// TIA Portal V18 export
// export: Created 2025-12-01T12:38:33.2765069Z, ExportSetting None, DisplayName Totally Integrated Automation Portal, DisplayVersion V18 Update 5, DisplayName TIA Portal Openness, DisplayVersion V18 Update 5, DisplayName TIA Portal Teamcenter Gateway, DisplayVersion V18, DisplayName TIA Portal Version Control Interface, DisplayVersion V18, DisplayName STEP 7 Professional, DisplayVersion V18 Update 5, DisplayName STEP 7 Safety, DisplayVersion V18, DisplayName WinCC Professional, DisplayVersion V18 Update 5
FUNCTION "ST10Cyl_interface1-10" : Void   // FC1020, LAD
{ S7_Optimized_Access := 'FALSE' }
// stored: AutoNumber false, SetENOAutomatically false
   VAR_INPUT
      AlwaysON : Bool;
      E_stop : Bool;
   END_VAR
   VAR_TEMP
      tTest : Bool;
      i : Int;
   END_VAR
BEGIN

REGION Network 1 (SCL): Cylinder 1-10 IO Interface (SCL)
   IF "Station_Sys".Manual.Mode THEN

       FOR #i := 1 TO 100 BY 1

       DO
           "ST10Cylinder".Cy[#i].In.ManualOutputType := TRUE;

       END_FOR;

   END_IF;

   //Cylinder1 IO  A-Loading-01HorizontalCylinder
   //Input
   "ST10Cylinder".Cy[1].In.WorkPositionSensor := "iA-Loading-01HorizontalCylinderInWP";
   "ST10Cylinder".Cy[1].In.HomePositionSensor := "iA-Loading-01HorizontalCylinderInHP";
   //Output
   "oA-Loading-01HorizontalCylinderToWP" := "ST10Cylinder".Cy[1].Out.GoWorkPosition;
   "oA-Loading-01HorizontalCylinderToHP" := "ST10Cylinder".Cy[1].Out.GoHomePosition;

   //Cylinder2 IO  A-Loading-01UpDownTakeCylinder
   //Input
   "ST10Cylinder".Cy[2].In.WorkPositionSensor := "iA-Loading-01UpDownTakeCylinderInWP";
   "ST10Cylinder".Cy[2].In.HomePositionSensor := "iA-Loading-01UpDownTakeCylinderInHP";
   //Output
   "oA-Loading-01UpDownTakeCylinderToWP" := "ST10Cylinder".Cy[2].Out.GoWorkPosition;
   "oA-Loading-01UpDownTakeCylinderToHP" := "ST10Cylinder".Cy[2].Out.GoHomePosition;

   //Cylinder3 IO  A-Loading-02HorizontalCylinder
   //Input
   "ST10Cylinder".Cy[3].In.WorkPositionSensor := "iA-Loading-02HorizontalCylinderInWP"  ;
   "ST10Cylinder".Cy[3].In.HomePositionSensor := "iA-Loading-02HorizontalCylinderInHP"  ;
   //Output
   "oA-Loading-02HorizontalCylinderToWP" := "ST10Cylinder".Cy[3].Out.GoWorkPosition;
   "oA-Loading-02HorizontalCylinderToHP" := "ST10Cylinder".Cy[3].Out.GoHomePosition;

   //Cylinder4 IO     A-Loading-02UpDownTakeCylinder
   //Input
   "ST10Cylinder".Cy[4].In.WorkPositionSensor := "iA-Loading-02UpDownTakeCylinderInWP";
   "ST10Cylinder".Cy[4].In.HomePositionSensor := "iA-Loading-02UpDownTakeCylinderInHP";
   //Output
   "oA-Loading-02UpDownTakeCylinderToWP" := "ST10Cylinder".Cy[4].Out.GoWorkPosition;
   "oA-Loading-02UpDownTakeCylinderToHP" := "ST10Cylinder".Cy[4].Out.GoHomePosition;

   //Cylinder5 IO  B-PressFitting-01GripperCylinder
   //Input
   "ST10Cylinder".Cy[5].In.WorkPositionSensor := "iB-PressFitting-01GripperCylinderInWP";
   "ST10Cylinder".Cy[5].In.HomePositionSensor := "iB-PressFitting-01GripperCylinderInHP";
   //Output
   "oB-PressFitting-01GripperCylinderToWP" := "ST10Cylinder".Cy[5].Out.GoWorkPosition;
   "oB-PressFitting-01GripperCylinderToHP" := "ST10Cylinder".Cy[5].Out.GoHomePosition;

   //Cylinder6 IO  B-PressFitting-01Cylinder
   //Input
   "ST10Cylinder".Cy[6].In.WorkPositionSensor := "iB-PressFitting-01CylinderInWP" ;
   "ST10Cylinder".Cy[6].In.HomePositionSensor := "iB-PressFitting-01CylinderInHP" ;
   //Output
   "oB-PressFitting-01CylinderToWP" := "ST10Cylinder".Cy[6].Out.GoWorkPosition;
   "oB-PressFitting-01CylinderToHP" := "ST10Cylinder".Cy[6].Out.GoHomePosition;

   //Cylinder7 IO  B-PressFitting-02GripperCylinder
   //Input
   "ST10Cylinder".Cy[7].In.WorkPositionSensor := "iB-PressFitting-02GripperCylinderInWP";
   "ST10Cylinder".Cy[7].In.HomePositionSensor := "iB-PressFitting-02GripperCylinderInHP";
   //Output
   "oB-PressFitting-02GripperCylinderToWP" := "ST10Cylinder".Cy[7].Out.GoWorkPosition;
   "oB-PressFitting-02GripperCylinderToHP" := "ST10Cylinder".Cy[7].Out.GoHomePosition;

   //Cylinder8 IO  B-PressFitting-02Cylinder
   //Input
   "ST10Cylinder".Cy[8].In.WorkPositionSensor := "iB-PressFitting-02CylinderInWP";
   "ST10Cylinder".Cy[8].In.HomePositionSensor := "iB-PressFitting-02CylinderInHP";
   //Output
   "oB-PressFitting-02CylinderToWP" := "ST10Cylinder".Cy[8].Out.GoWorkPosition;
   "oB-PressFitting-02CylinderToHP" := "ST10Cylinder".Cy[8].Out.GoHomePosition;

   //Cylinder9 IO  C-LocationCylinder
   //Input
   "ST10Cylinder".Cy[9].In.WorkPositionSensor := "iC-LocationCylinderInWP";
   "ST10Cylinder".Cy[9].In.HomePositionSensor := "iC-LocationCylinderInHP";
   //Output
   "oC-LocationCylinderToWP" := "ST10Cylinder".Cy[9].Out.GoWorkPosition;
   "oC-LocationCylinderToHP" := "ST10Cylinder".Cy[9].Out.GoHomePosition;


   //Cylinder10 IO  Spare
   //Input
   "ST10Cylinder".Cy[10].In.WorkPositionSensor := "ST10Cylinder".Cy[10].Out.GoWorkPosition ;
   "ST10Cylinder".Cy[10].In.HomePositionSensor := "ST10Cylinder".Cy[10].Out.GoHomePosition ;
   //Output
   "ST10Cylinder".Cy[10].Out.GoWorkPosition := "ST10Cylinder".Cy[10].Out.GoWorkPosition;
   "ST10Cylinder".Cy[10].Out.GoHomePosition := "ST10Cylinder".Cy[10].Out.GoHomePosition;
END_REGION

REGION Network 2: CY1 interface A-Loading-01HorizontalCylinder
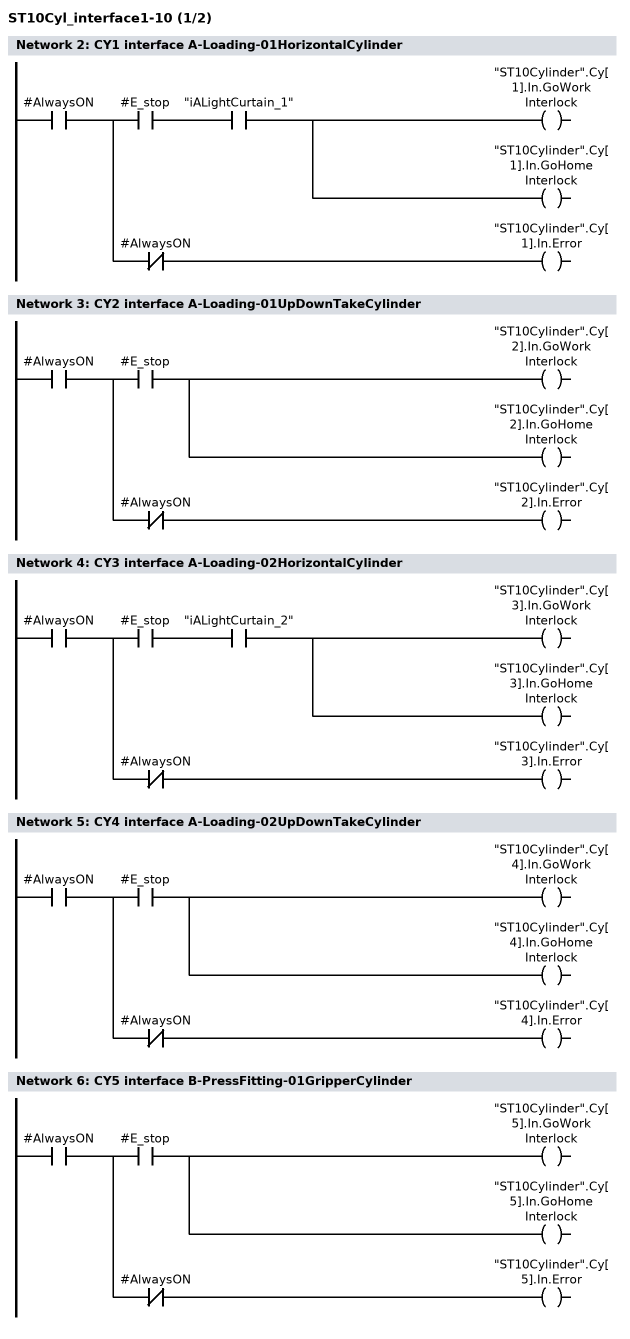
   RUNG wire#powerrail
      Contact( #AlwaysON )
      wire#w1
      Contact( #E_stop )
      Contact( "iALightCurtain_1" )
      wire#w2
      Coil( "ST10Cylinder".Cy[1].In.GoWorkInterlock )
   END_RUNG
   RUNG wire#w2
      Coil( "ST10Cylinder".Cy[1].In.GoHomeInterlock )
   END_RUNG
   RUNG wire#w1
      I_Contact( #AlwaysON )
      Coil( "ST10Cylinder".Cy[1].In.Error )
   END_RUNG
   // the same network as SCL:
   "ST10Cylinder".Cy[1].In.GoWorkInterlock := #AlwaysON AND #E_stop AND "iALightCurtain_1";
   "ST10Cylinder".Cy[1].In.GoHomeInterlock := #AlwaysON AND #E_stop AND "iALightCurtain_1";
   "ST10Cylinder".Cy[1].In.Error := #AlwaysON AND NOT #AlwaysON;
END_REGION

REGION Network 3: CY2 interface A-Loading-01UpDownTakeCylinder
   RUNG wire#powerrail
      Contact( #AlwaysON )
      wire#w1
      Contact( #E_stop )
      wire#w2
      Coil( "ST10Cylinder".Cy[2].In.GoWorkInterlock )
   END_RUNG
   RUNG wire#w2
      Coil( "ST10Cylinder".Cy[2].In.GoHomeInterlock )
   END_RUNG
   RUNG wire#w1
      I_Contact( #AlwaysON )
      Coil( "ST10Cylinder".Cy[2].In.Error )
   END_RUNG
   // the same network as SCL:
   "ST10Cylinder".Cy[2].In.GoWorkInterlock := #AlwaysON AND #E_stop;
   "ST10Cylinder".Cy[2].In.GoHomeInterlock := #AlwaysON AND #E_stop;
   "ST10Cylinder".Cy[2].In.Error := #AlwaysON AND NOT #AlwaysON;
END_REGION

REGION Network 4: CY3 interface A-Loading-02HorizontalCylinder
   RUNG wire#powerrail
      Contact( #AlwaysON )
      wire#w1
      Contact( #E_stop )
      Contact( "iALightCurtain_2" )
      wire#w2
      Coil( "ST10Cylinder".Cy[3].In.GoWorkInterlock )
   END_RUNG
   RUNG wire#w2
      Coil( "ST10Cylinder".Cy[3].In.GoHomeInterlock )
   END_RUNG
   RUNG wire#w1
      I_Contact( #AlwaysON )
      Coil( "ST10Cylinder".Cy[3].In.Error )
   END_RUNG
   // the same network as SCL:
   "ST10Cylinder".Cy[3].In.GoWorkInterlock := #AlwaysON AND #E_stop AND "iALightCurtain_2";
   "ST10Cylinder".Cy[3].In.GoHomeInterlock := #AlwaysON AND #E_stop AND "iALightCurtain_2";
   "ST10Cylinder".Cy[3].In.Error := #AlwaysON AND NOT #AlwaysON;
END_REGION

REGION Network 5: CY4 interface A-Loading-02UpDownTakeCylinder
   RUNG wire#powerrail
      Contact( #AlwaysON )
      wire#w1
      Contact( #E_stop )
      wire#w2
      Coil( "ST10Cylinder".Cy[4].In.GoWorkInterlock )
   END_RUNG
   RUNG wire#w2
      Coil( "ST10Cylinder".Cy[4].In.GoHomeInterlock )
   END_RUNG
   RUNG wire#w1
      I_Contact( #AlwaysON )
      Coil( "ST10Cylinder".Cy[4].In.Error )
   END_RUNG
   // the same network as SCL:
   "ST10Cylinder".Cy[4].In.GoWorkInterlock := #AlwaysON AND #E_stop;
   "ST10Cylinder".Cy[4].In.GoHomeInterlock := #AlwaysON AND #E_stop;
   "ST10Cylinder".Cy[4].In.Error := #AlwaysON AND NOT #AlwaysON;
END_REGION

REGION Network 6: CY5 interface B-PressFitting-01GripperCylinder
   RUNG wire#powerrail
      Contact( #AlwaysON )
      wire#w1
      Contact( #E_stop )
      wire#w2
      Coil( "ST10Cylinder".Cy[5].In.GoWorkInterlock )
   END_RUNG
   RUNG wire#w2
      Coil( "ST10Cylinder".Cy[5].In.GoHomeInterlock )
   END_RUNG
   RUNG wire#w1
      I_Contact( #AlwaysON )
      Coil( "ST10Cylinder".Cy[5].In.Error )
   END_RUNG
   // the same network as SCL:
   "ST10Cylinder".Cy[5].In.GoWorkInterlock := #AlwaysON AND #E_stop;
   "ST10Cylinder".Cy[5].In.GoHomeInterlock := #AlwaysON AND #E_stop;
   "ST10Cylinder".Cy[5].In.Error := #AlwaysON AND NOT #AlwaysON;
END_REGION

REGION Network 7: CY6 interface B-PressFitting-01Cylinder
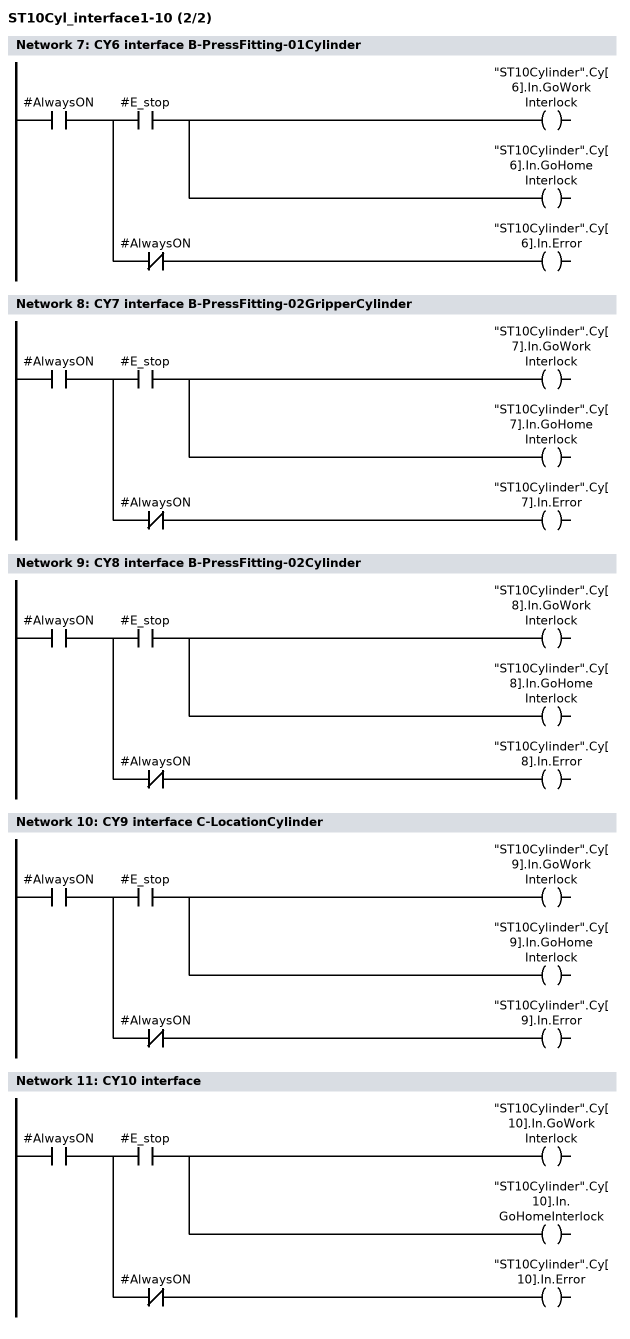
   RUNG wire#powerrail
      Contact( #AlwaysON )
      wire#w1
      Contact( #E_stop )
      wire#w2
      Coil( "ST10Cylinder".Cy[6].In.GoWorkInterlock )
   END_RUNG
   RUNG wire#w2
      Coil( "ST10Cylinder".Cy[6].In.GoHomeInterlock )
   END_RUNG
   RUNG wire#w1
      I_Contact( #AlwaysON )
      Coil( "ST10Cylinder".Cy[6].In.Error )
   END_RUNG
   // the same network as SCL:
   "ST10Cylinder".Cy[6].In.GoWorkInterlock := #AlwaysON AND #E_stop;
   "ST10Cylinder".Cy[6].In.GoHomeInterlock := #AlwaysON AND #E_stop;
   "ST10Cylinder".Cy[6].In.Error := #AlwaysON AND NOT #AlwaysON;
END_REGION

REGION Network 8: CY7 interface B-PressFitting-02GripperCylinder
   RUNG wire#powerrail
      Contact( #AlwaysON )
      wire#w1
      Contact( #E_stop )
      wire#w2
      Coil( "ST10Cylinder".Cy[7].In.GoWorkInterlock )
   END_RUNG
   RUNG wire#w2
      Coil( "ST10Cylinder".Cy[7].In.GoHomeInterlock )
   END_RUNG
   RUNG wire#w1
      I_Contact( #AlwaysON )
      Coil( "ST10Cylinder".Cy[7].In.Error )
   END_RUNG
   // the same network as SCL:
   "ST10Cylinder".Cy[7].In.GoWorkInterlock := #AlwaysON AND #E_stop;
   "ST10Cylinder".Cy[7].In.GoHomeInterlock := #AlwaysON AND #E_stop;
   "ST10Cylinder".Cy[7].In.Error := #AlwaysON AND NOT #AlwaysON;
END_REGION

REGION Network 9: CY8 interface B-PressFitting-02Cylinder
   RUNG wire#powerrail
      Contact( #AlwaysON )
      wire#w1
      Contact( #E_stop )
      wire#w2
      Coil( "ST10Cylinder".Cy[8].In.GoWorkInterlock )
   END_RUNG
   RUNG wire#w2
      Coil( "ST10Cylinder".Cy[8].In.GoHomeInterlock )
   END_RUNG
   RUNG wire#w1
      I_Contact( #AlwaysON )
      Coil( "ST10Cylinder".Cy[8].In.Error )
   END_RUNG
   // the same network as SCL:
   "ST10Cylinder".Cy[8].In.GoWorkInterlock := #AlwaysON AND #E_stop;
   "ST10Cylinder".Cy[8].In.GoHomeInterlock := #AlwaysON AND #E_stop;
   "ST10Cylinder".Cy[8].In.Error := #AlwaysON AND NOT #AlwaysON;
END_REGION

REGION Network 10: CY9 interface C-LocationCylinder
   RUNG wire#powerrail
      Contact( #AlwaysON )
      wire#w1
      Contact( #E_stop )
      wire#w2
      Coil( "ST10Cylinder".Cy[9].In.GoWorkInterlock )
   END_RUNG
   RUNG wire#w2
      Coil( "ST10Cylinder".Cy[9].In.GoHomeInterlock )
   END_RUNG
   RUNG wire#w1
      I_Contact( #AlwaysON )
      Coil( "ST10Cylinder".Cy[9].In.Error )
   END_RUNG
   // the same network as SCL:
   "ST10Cylinder".Cy[9].In.GoWorkInterlock := #AlwaysON AND #E_stop;
   "ST10Cylinder".Cy[9].In.GoHomeInterlock := #AlwaysON AND #E_stop;
   "ST10Cylinder".Cy[9].In.Error := #AlwaysON AND NOT #AlwaysON;
END_REGION

REGION Network 11: CY10 interface
   RUNG wire#powerrail
      Contact( #AlwaysON )
      wire#w1
      Contact( #E_stop )
      wire#w2
      Coil( "ST10Cylinder".Cy[10].In.GoWorkInterlock )
   END_RUNG
   RUNG wire#w2
      Coil( "ST10Cylinder".Cy[10].In.GoHomeInterlock )
   END_RUNG
   RUNG wire#w1
      I_Contact( #AlwaysON )
      Coil( "ST10Cylinder".Cy[10].In.Error )
   END_RUNG
   // the same network as SCL:
   "ST10Cylinder".Cy[10].In.GoWorkInterlock := #AlwaysON AND #E_stop;
   "ST10Cylinder".Cy[10].In.GoHomeInterlock := #AlwaysON AND #E_stop;
   "ST10Cylinder".Cy[10].In.Error := #AlwaysON AND NOT #AlwaysON;
END_REGION
END_FUNCTION
